(* CoDeSys 2.3 library: SysLibTargetVisu.lib *)

(* Global variable list: Globale_Variablen *)
VAR_GLOBAL CONSTANT
	DF_LEFT: WORD := 16#0001;
	DF_RIGHT: WORD := 16#0002;
	DF_HCENTER: WORD := 16#0004;
	DF_TOP: WORD := 16#0008;
	DF_BOTTOM: WORD := 16#0010;
	DF_VCENTER: WORD := 16#0020;

	FF_ITALIC: WORD :=16#0001;
	FF_BOLD: WORD :=16#0002;
	FF_UNDERLINED: WORD :=16#0004;
	FF_STRIKEDOUT: WORD :=16#0008;

	FF_SOLID:  WORD := 16#0000;
	FF_NULL: WORD := 16#0001;

	LF_SOLID:  WORD:= 16#0000;
	LF_NULL: WORD := 16#0001;

	DC_WHITE: DWORD := 16#00_FF_FF_FF;
	DC_BLACK: DWORD := 16#00_00_00_00;
	NUMOFUSERS:INT:=7; (*0..7*)
END_VAR
VAR_GLOBAL
	RTGraphic_PB:POINTER TO BOOL;
	RTGraphic_PC:POINTER TO BOOL;
	RTGraphic_Text:STRING(256);
	RTGraphic_VisuScaleINT:INT := 1000;
	RTGraphic_VisuPositionXINT:INT := 0;
	RTGraphic_VisuPositionYINT:INT := 0;
	RTGraphic_MotherVisuString:STRING;
	RTGraphic_ChildVisuString:STRING;
	RTGraphic_ResBool:BOOL;
	RTGraphic_CountDWORD:DWORD;
	RTGraphic_ButtonIsClicked:BOOL;
	(* Variables for input task *)
	RTGraphic_Input_String:STRING(256);
	RTGraphic_Input_CenterX:INT;
	RTGraphic_Input_CenterY:INT;
	RTGraphic_Input_nX:INT;
	RTGraphic_Input_nY:INT;
	RTGraphic_Input_RectLeft:INT;
	RTGraphic_Input_RectTop:INT;
	RTGraphic_Input_RectRight:INT;
	RTGraphic_Input_RectBottom:INT;
	RTGraphic_IsClicked:SINT;
	RTGraphic_Input_dw:DWORD;
	RTGraphic_Input_di:DINT;
	RTGraphic_Input_lr:LREAL;
      (* Variables for paint task *)
	RTGraphic_String:STRING(256);
	RTGraphic_CenterX:INT;
	RTGraphic_CenterY:INT;
	RTGraphic_nX:INT;
	RTGraphic_nY:INT;
	RTGraphic_RectLeft:INT;
	RTGraphic_RectTop:INT;
	RTGraphic_RectRight:INT;
	RTGraphic_RectBottom:INT;
	RTGraphic_dw:DWORD;
	RTGraphic_di:DINT;
	RTGraphic_lr:LREAL;
END_VAR

(* Data type *)
TYPE Bitmap :
STRUCT
	 bmType:DINT;
    	 bmWidth:DINT;
   	 bmHeight:DINT;
   	 bmWidthBytes:DINT;
	 bmPlanes:INT;
	 bmBitsPixel:INT;
 	 bmBits:POINTER TO BYTE;
END_STRUCT
END_TYPE

(* POU BeginPaint, ST *)
FUNCTION BeginPaint : BOOL
VAR_INPUT
	stName: STRING;
	dwFlags:DWORD;
	nBmpId:INT;
	dwBgColor:DWORD;
END_VAR
;
END_FUNCTION

(* POU CalcRotation, ST *)
FUNCTION CalcRotation : BOOL
VAR_INPUT
	pnXCorner:POINTER TO INT;
	pnYCorner:POINTER TO INT;
	pmXCorner:POINTER TO INT;
	pmYCorner:POINTER TO INT;
	nXCenter:INT;
	nYCenter:INT;
	nAngle:DINT;
END_VAR
;
END_FUNCTION

(* POU ChangePassword, ST *)
FUNCTION ChangePassword : BOOL
VAR_INPUT
	pCurrentUserLevel:POINTER TO INT;
	nCurrentNumOfUsers:INT;
	pCurrentUsers:POINTER TO ARRAY [0..NUMOFUSERS] OF STRING;
	pCurrentPasswords:POINTER TO ARRAY [0..NUMOFUSERS] OF STRING;
	pCurrentLevels:POINTER TO ARRAY [0..NUMOFUSERS] OF INT;
END_VAR
;
END_FUNCTION

(* POU ChangeUserLevel, ST *)
FUNCTION ChangeUserLevel : BOOL
VAR_INPUT
	pCurrentUserLevel:POINTER TO INT;
	nCurrentNumOfUsers:INT;
       pCurrentUsers:POINTER TO ARRAY [0..NUMOFUSERS] OF STRING;
	pCurrentPasswords:POINTER TO ARRAY [0..NUMOFUSERS] OF STRING;
	pCurrentLevels:POINTER TO ARRAY [0..NUMOFUSERS] OF INT;
END_VAR
;
END_FUNCTION

(* POU CreateBitmap, ST *)
FUNCTION CreateBitmap : INT
VAR_INPUT
	nSize:DINT;
	pdwBitmap:POINTER TO DWORD;
END_VAR
;
END_FUNCTION

(* POU CreateUserdefinedControl, ST *)
FUNCTION CreateUserdefinedControl : INT
VAR_INPUT
	stIdentification : STRING(256);
	stParams : STRING(256);
	iType : INT;
END_VAR
VAR
END_VAR
;
END_FUNCTION

(* POU DeleteBitmap, ST *)
FUNCTION DeleteBitmap : BOOL
VAR_INPUT
	nId:INT;
END_VAR
;
END_FUNCTION

(* POU DrawBitmap, ST *)
FUNCTION DrawBitmap : BOOL
VAR_INPUT
	nId:INT;
	nXCorner:INT;
	nYCorner:INT;
	mXCorner:INT;
	mYCorner:INT;
	nIso:INT;
	dwColorTransparent:DWORD;
	bVisible:BOOL;
END_VAR
;
END_FUNCTION

(* POU DrawBitmapByString, ST *)
FUNCTION DrawBitmapByString : BOOL
VAR_INPUT
	stBitmap:STRING;
	nXCorner:INT;
	nYCorner:INT;
	mXCorner:INT;
	mYCorner:INT;
	nIso:INT;
	dwColorTransparent:DWORD;
	bVisible:BOOL;
END_VAR
;
END_FUNCTION

(* POU DrawButton, ST *)
FUNCTION DrawButton : BOOL
VAR_INPUT
	nXCorner:INT;
	nYCorner:INT;
	mXCorner:INT;
	mYCorner:INT;
	stText:STRING(256);
	dwDrawFlags:DWORD;
	bIsClicked:BOOL;
	dwFlags:DWORD;
	bVisible:BOOL;
END_VAR
;
END_FUNCTION

(* POU DrawEditC, ST *)
FUNCTION DrawEditC : BOOL
VAR_INPUT
	nXCorner:INT;
	nYCorner:INT;
	mXCorner:INT;
	mYCorner:INT;
	stText:STRING(256);
	stExpression:STRING;
	nIsString:INT;
	nType:INT;
	stMin:STRING;
	stMax:STRING;
	stComment:STRING;
END_VAR
;
END_FUNCTION

(* POU DrawPie, ST *)
FUNCTION DrawPie : BOOL
VAR_INPUT
	nXCorner:INT;
	nYCorner:INT;
	mXCorner:INT;
	mYCorner:INT;
	nAngleStart:INT;
	nAngleEnd:INT;
	nAngle:DINT;
	dwPieFlags:DWORD;
	stText:STRING(256);
	dwDrawFlags:DWORD;
	bVisible:BOOL;
END_VAR
VAR
END_VAR
;
END_FUNCTION

(* POU DrawPolygon, ST *)
FUNCTION DrawPolygon : BOOL
VAR_INPUT
	nNumberOfPoints:INT;
	pnXPoints:POINTER TO INT;
	pnYPoints:POINTER TO INT;
	stText:STRING(256);
	dwDrawFlags:DWORD;
	nType:INT;
	bVisible:BOOL;
END_VAR
;
END_FUNCTION

(* POU DrawRect, ST *)
FUNCTION DrawRect : BOOL
VAR_INPUT
	nXCorner:INT;
	nYCorner:INT;
	mXCorner:INT;
	mYCorner:INT;
	stText:STRING(256);
	dwDrawFlags:DWORD;
	nType:INT;
	bVisible:BOOL;
END_VAR
;
END_FUNCTION

(* POU DrawText, ST *)
FUNCTION DrawText : BOOL
VAR_INPUT
	nXCorner:INT;
	nYCorner:INT;
	mXCorner:INT;
	mYCorner:INT;
	stText:STRING(256);
	dwDrawFlags:DWORD;
	bVisible:BOOL;
END_VAR
;
END_FUNCTION

(* POU EndPaint, ST *)
FUNCTION EndPaint : BOOL
VAR_INPUT
	stName: STRING;
	dwFlags:DWORD;
END_VAR
;
END_FUNCTION

(* POU EnumToString, ST *)
FUNCTION EnumToString : BOOL
VAR_INPUT
	nId:INT;
	pstEnum:POINTER TO STRING;
	nEnum:INT;
END_VAR
;
END_FUNCTION

(* POU ExecuteCommand, ST *)
FUNCTION ExecuteCommand : SINT
VAR_INPUT
	stCommand:STRING(1024);
	nType:INT;
END_VAR
;
END_FUNCTION

(* POU ExecuteUserdefinedControlCall, ST *)
FUNCTION ExecuteUserdefinedControlCall : BOOL
VAR_INPUT
	nIndex : INT;
	stCallIdentification : STRING(256);
	stParam : STRING(256);
	pstReturnValue : POINTER TO STRING(256);			(* may be null if no return value is expected *)
	nReturnBufferSize : INT;									(* the maximal number of characters that can be returned in pstReturnValue *)
	pbValueReturned : POINTER TO BOOL;					(* may be null if no return value is expected *)
END_VAR
VAR
END_VAR
;
END_FUNCTION

(* POU GetSurroundRect, ST *)
FUNCTION GetSurroundRect : BOOL
VAR_INPUT
	pnXCorner:POINTER TO INT;
	pnYCorner:POINTER TO INT;
	pmXCorner:POINTER TO INT;
	pmYCorner:POINTER TO INT;
	nNumberOfPoints:INT;
	pnXPoints:POINTER TO INT;
	pnYPoints:POINTER TO INT;
END_VAR
;
END_FUNCTION

(* POU GetText, ST *)
FUNCTION GetText : BOOL
VAR_INPUT
	stResult: STRING(256);
	nResultLength:INT;
	stPrefix: STRING;
	dwID: DWORD;
END_VAR
;
END_FUNCTION

(* POU GetTextByStringId, ST *)
FUNCTION GetTextByStringId : BOOL
VAR_INPUT
	stResult: STRING(256);
	nResultLength:INT;
	stPrefix: STRING;
	stID: STRING;
END_VAR
;
END_FUNCTION

(* POU GetUnicodeText, ST *)
FUNCTION GetUnicodeText : BOOL
VAR_INPUT
	pResult: POINTER TO ARRAY[0..10000] OF UINT;
	nResultLength:INT;
	stPrefix: STRING;
	dwID: DWORD;
END_VAR
;
END_FUNCTION

(* POU GetUnicodeTextByStringId, ST *)
FUNCTION GetUnicodeTextByStringId : BOOL
VAR_INPUT
	pResult: POINTER TO ARRAY[0..10000] OF UINT;
	nResultLength:INT;
	stPrefix: STRING;
	stID: STRING;
END_VAR
;
END_FUNCTION

(* POU IsClickedEditC, ST *)
FUNCTION IsClickedEditC : BOOL
VAR_INPUT
	nXCorner:INT;
	nYCorner:INT;
	mXCorner:INT;
	mYCorner:INT;
	bUp:BOOL;
	bToggle:BOOL;
	bVisible:BOOL;
END_VAR
;
END_FUNCTION

(* POU IsClickedPolygon, ST *)
FUNCTION IsClickedPolygon : SINT
VAR_INPUT
	nNumberOfPoints:INT;
	pnXPoints:POINTER TO INT;
	pnYPoints:POINTER TO INT;
	bUp:BOOL;
	bToggle:BOOL;
	nType:INT;
	bVisible:BOOL;
END_VAR
;
END_FUNCTION

(* POU IsClickedRect, ST *)
FUNCTION IsClickedRect : SINT
VAR_INPUT
	nXCorner:INT;
	nYCorner:INT;
	mXCorner:INT;
	mYCorner:INT;
	bUp:BOOL;
	bToggle:BOOL;
	nType:INT;
	bVisible:BOOL;
END_VAR
;
END_FUNCTION

(* POU IsClosedEditC, ST *)
FUNCTION IsClosedEditC : BOOL
VAR_INPUT
	stExpression:STRING;
END_VAR
;
END_FUNCTION

(* POU IsKeyPressed, ST *)
FUNCTION IsKeyPressed : BOOL
VAR_INPUT
	nKeyCode:INT;
	bUp:BOOL;
	nInfo:INT;
END_VAR
VAR
END_VAR
;
END_FUNCTION

(* POU IsMovedInPolygon, ST *)
FUNCTION IsMovedInPolygon : SINT
VAR_INPUT
	nNumberOfPoints:INT;
	pnXPoints:POINTER TO INT;
	pnYPoints:POINTER TO INT;
	pnX:POINTER TO INT;
	pnY:POINTER TO INT;
	nType:INT;
	bVisible:BOOL;
END_VAR
;
END_FUNCTION

(* POU IsMovedInRect, ST *)
FUNCTION IsMovedInRect : SINT
VAR_INPUT
	nXCorner:INT;
	nYCorner:INT;
	mXCorner:INT;
	mYCorner:INT;
	pnX:POINTER TO INT;
	pnY:POINTER TO INT;
	nType:INT;
	bVisible:BOOL;
END_VAR
;
END_FUNCTION

(* POU MovePolygon, ST *)
FUNCTION MovePolygon : BOOL
VAR_INPUT
	nNumberOfPoints:INT;
	pnXPoints:POINTER TO INT;
	pnYPoints:POINTER TO INT;
	nXCenter:INT;
	nYCenter:INT;
	nScale:DINT;
	nAngle:DINT;
	nXOffset:DINT;
	nYOffset:DINT;
END_VAR
;
END_FUNCTION

(* POU PopTransformation, ST *)
FUNCTION PopTransformation : BOOL
VAR_INPUT
	mXmother:INT;
	mYmother:INT;
	nXChild:INT;
	nYChild:INT;
	mXChild:INT;
	mYChild:INT;
	bIso:BOOL;
	bClipFrame:BOOL;
END_VAR
VAR
END_VAR
;
END_FUNCTION

(* POU Printf, ST *)
FUNCTION Printf : STRING(256)
VAR_INPUT
	stFormat: STRING;
	dwValue: POINTER TO BYTE;
	nType: INT;
END_VAR
;
END_FUNCTION

(* POU PrintfInput, ST *)
FUNCTION PrintfInput : STRING(256)
VAR_INPUT
	stFormat: STRING;
	dwValue: POINTER TO BYTE;
	nType: INT;
END_VAR
;
END_FUNCTION

(* POU PushTransformation, ST *)
FUNCTION PushTransformation : BOOL
VAR_INPUT
	mXmother:INT;
	mYmother:INT;
	nXChild:INT;
	nYChild:INT;
	mXChild:INT;
	mYChild:INT;
	bIso:BOOL;
	bClipFrame:BOOL;
END_VAR
VAR
END_VAR
;
END_FUNCTION

(* POU RefreshUserdefinedControl, ST *)
FUNCTION RefreshUserdefinedControl : BOOL
VAR_INPUT
	nIndex : INT;
	nXCorner : INT;
	nYCorner : INT;
	mXCorner : INT;
	mYCorner : INT;
	bVisible : BOOL;
END_VAR
VAR
END_VAR
;
END_FUNCTION

(* POU RegisterVariable, ST *)
FUNCTION RegisterVariable : BOOL
VAR_INPUT
	stName: STRING;
	stValue: STRING;
	stAdr:STRING;
	nType: INT;
END_VAR
;
END_FUNCTION

(* POU ReturnEnteredValue, ST *)
FUNCTION ReturnEnteredValue :STRING(256)
VAR_INPUT
	stExpression:STRING;
END_VAR
;
END_FUNCTION

(* POU RGBColor, ST *)
FUNCTION RGBColor : DINT
VAR_INPUT
	byRed: BYTE;
	byGreen: BYTE;
	byBlue: BYTE;
END_VAR
;
END_FUNCTION

(* POU SendBitmap, ST *)
FUNCTION SendBitmap : INT
VAR_INPUT
	stFile:STRING;
END_VAR
;
END_FUNCTION

(* POU SendEnum, ST *)
FUNCTION SendEnum : INT
VAR_INPUT
	stDescription:STRING;
END_VAR
;
END_FUNCTION

(* POU SetFill, ST *)
FUNCTION SetFill : BOOL
VAR_INPUT
	dwFillFlags:DWORD;
	dwFillColor:DWORD;
END_VAR
;
END_FUNCTION

(* POU SetFont, ST *)
FUNCTION SetFont : BOOL
VAR_INPUT
	stFontName:STRING;
	nFontSize:INT;
	dwFontFlags:DWORD;
	dwFontColor:DWORD;
END_VAR
;
END_FUNCTION

(* POU SetLine, ST *)
FUNCTION SetLine : BOOL
VAR_INPUT
	nBorderWidth:INT;
	dwBorderFlags:DWORD;
	dwBorderColor:DWORD;
END_VAR
;
END_FUNCTION

(* POU StopVisu, ST *)
FUNCTION StopVisu : BOOL
VAR_INPUT
	stName: STRING;
END_VAR
;
END_FUNCTION

(* POU StringToEnum, ST *)
FUNCTION StringToEnum : BOOL
VAR_INPUT
	nId:INT;
	nEnum:POINTER TO INT;
	stEnum:STRING;
END_VAR
;
END_FUNCTION

(* POU TransformPoint, ST *)
(* This function executes the transformation for coordinates to the currently active transformation or backwards *)
FUNCTION TransformPoint : BOOL
VAR_INPUT
	px : POINTER TO INT;				(* This parameter points to the x coordinate that shall be transformed. This value will be changed during the call! *)
	py : POINTER TO INT;				(* This parameter points to the y coordinate that shall be transformed. This value will be changed during the call! *)
	bTransform : BOOL;				(* This parameter decides the transformation direction, TRUE will transform the point into the currently
											active transformation, FALSE will transform a point outof the actual transformation. This means
											TRUE will transform a client point to a screen coordinate, FALSE a screen point to a client point where a
											client point is a point in the local coordinate system of the active reference. *)
	dwFlags : DWORD;				(* This parameter is reservered. Must be 0 *)
END_VAR
VAR
END_VAR
;
END_FUNCTION

(* POU Version2326, ST *)
FUNCTION Version2326 : BOOL
VAR_INPUT
	Version:INT;
END_VAR
VAR
END_VAR
;
END_FUNCTION
